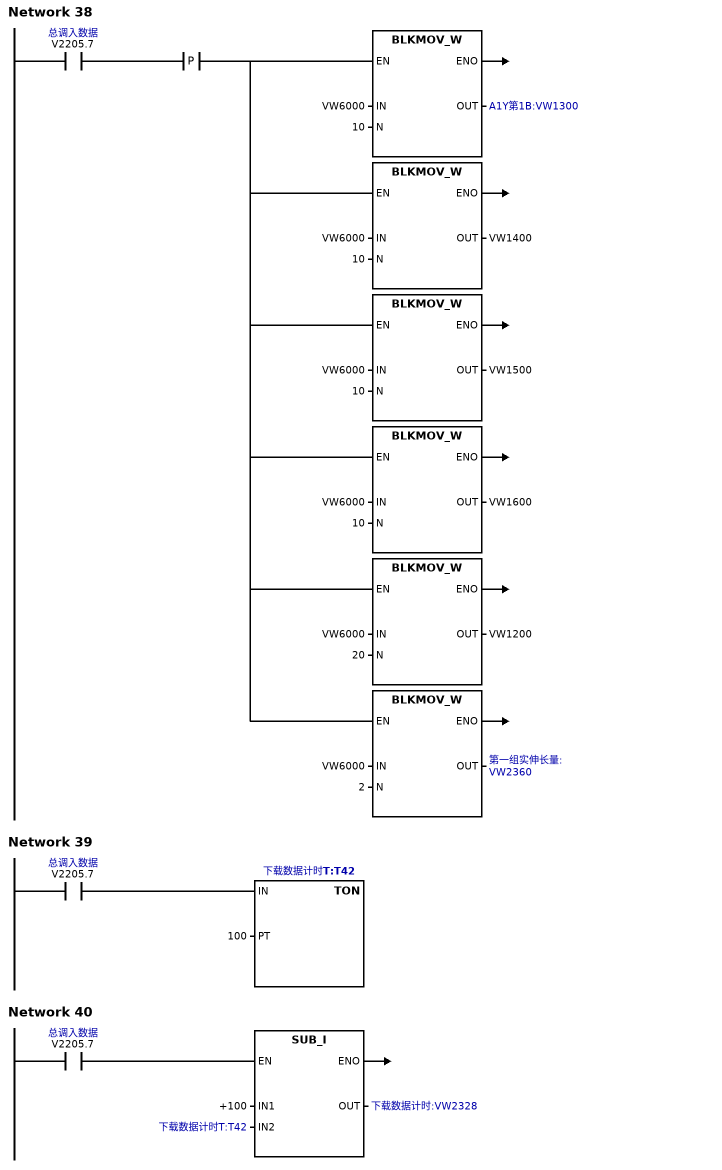
[picture p48: SBR18 networks 38-40]
Network 38
LD     总调入数据:V2205.7
EU
BMW    VW6000, A1Y第1B:VW1300, 10
BMW    VW6000, VW1400, 10
BMW    VW6000, VW1500, 10
BMW    VW6000, VW1600, 10
BMW    VW6000, VW1200, 20
BMW    VW6000, 第一组实伸长量:VW2360, 2
Network 39
LD     总调入数据:V2205.7
TON    下载数据计时T:T42, 100
Network 40
LD     总调入数据:V2205.7
MOVW   +100, 下载数据计时:VW2328
-I     下载数据计时T:T42, 下载数据计时:VW2328
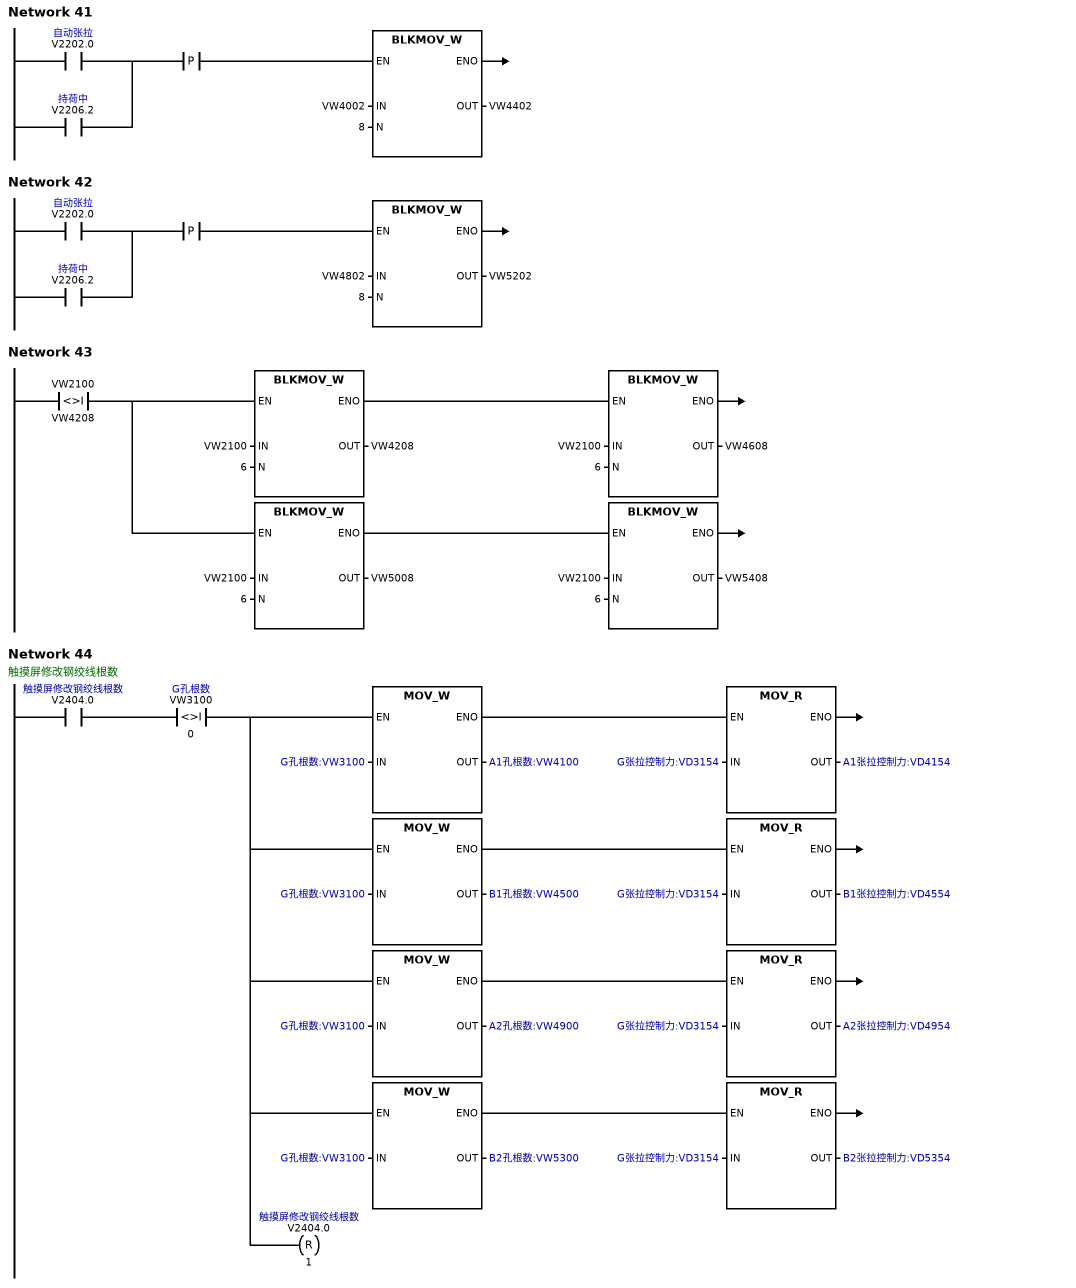
Network 41
LD     自动张拉:V2202.0
O      持荷中:V2206.2
EU
BMW    VW4002, VW4402, 8
Network 42
LD     自动张拉:V2202.0
O      持荷中:V2206.2
EU
BMW    VW4802, VW5202, 8
Network 43
LDW<>  VW2100, VW4208
LPS
BMW    VW2100, VW4208, 6
AENO
BMW    VW2100, VW4608, 6
LPP
BMW    VW2100, VW5008, 6
AENO
BMW    VW2100, VW5408, 6
Network 44
// 触摸屏修改钢绞线根数
LD     触摸屏修改钢绞线根数:V2404.0
AW<>   G孔根数:VW3100, 0
LPS
MOVW   G孔根数:VW3100, A1孔根数:VW4100
AENO
MOVR   G张拉控制力:VD3154, A1张拉控制力:VD4154
LRD
MOVW   G孔根数:VW3100, B1孔根数:VW4500
AENO
MOVR   G张拉控制力:VD3154, B1张拉控制力:VD4554
LRD
MOVW   G孔根数:VW3100, A2孔根数:VW4900
AENO
MOVR   G张拉控制力:VD3154, A2张拉控制力:VD4954
LRD
MOVW   G孔根数:VW3100, B2孔根数:VW5300
AENO
MOVR   G张拉控制力:VD3154, B2张拉控制力:VD5354
LPP
R      触摸屏修改钢绞线根数:V2404.0, 1
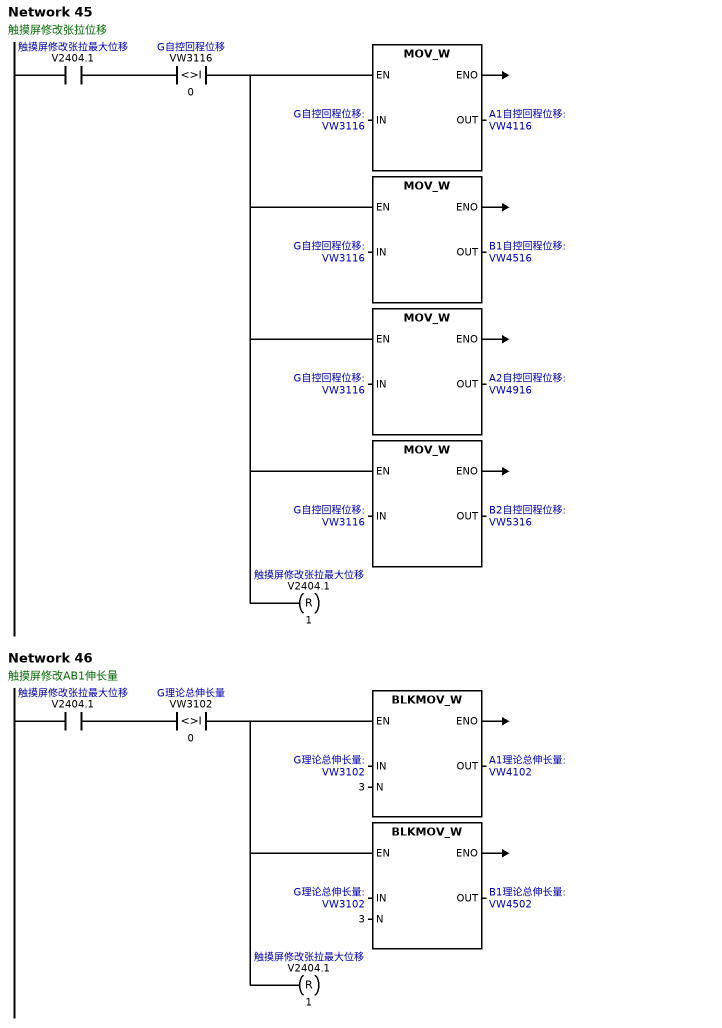
Network 45
// 触摸屏修改张拉位移
LD     触摸屏修改张拉最大位移:V2404.1
AW<>   G自控回程位移:VW3116, 0
MOVW   G自控回程位移:VW3116, A1自控回程位移:VW4116
MOVW   G自控回程位移:VW3116, B1自控回程位移:VW4516
MOVW   G自控回程位移:VW3116, A2自控回程位移:VW4916
MOVW   G自控回程位移:VW3116, B2自控回程位移:VW5316
R      触摸屏修改张拉最大位移:V2404.1, 1
Network 46
// 触摸屏修改AB1伸长量
LD     触摸屏修改张拉最大位移:V2404.1
AW<>   G理论总伸长量:VW3102, 0
BMW    G理论总伸长量:VW3102, A1理论总伸长量:VW4102, 3
BMW    G理论总伸长量:VW3102, B1理论总伸长量:VW4502, 3
R      触摸屏修改张拉最大位移:V2404.1, 1
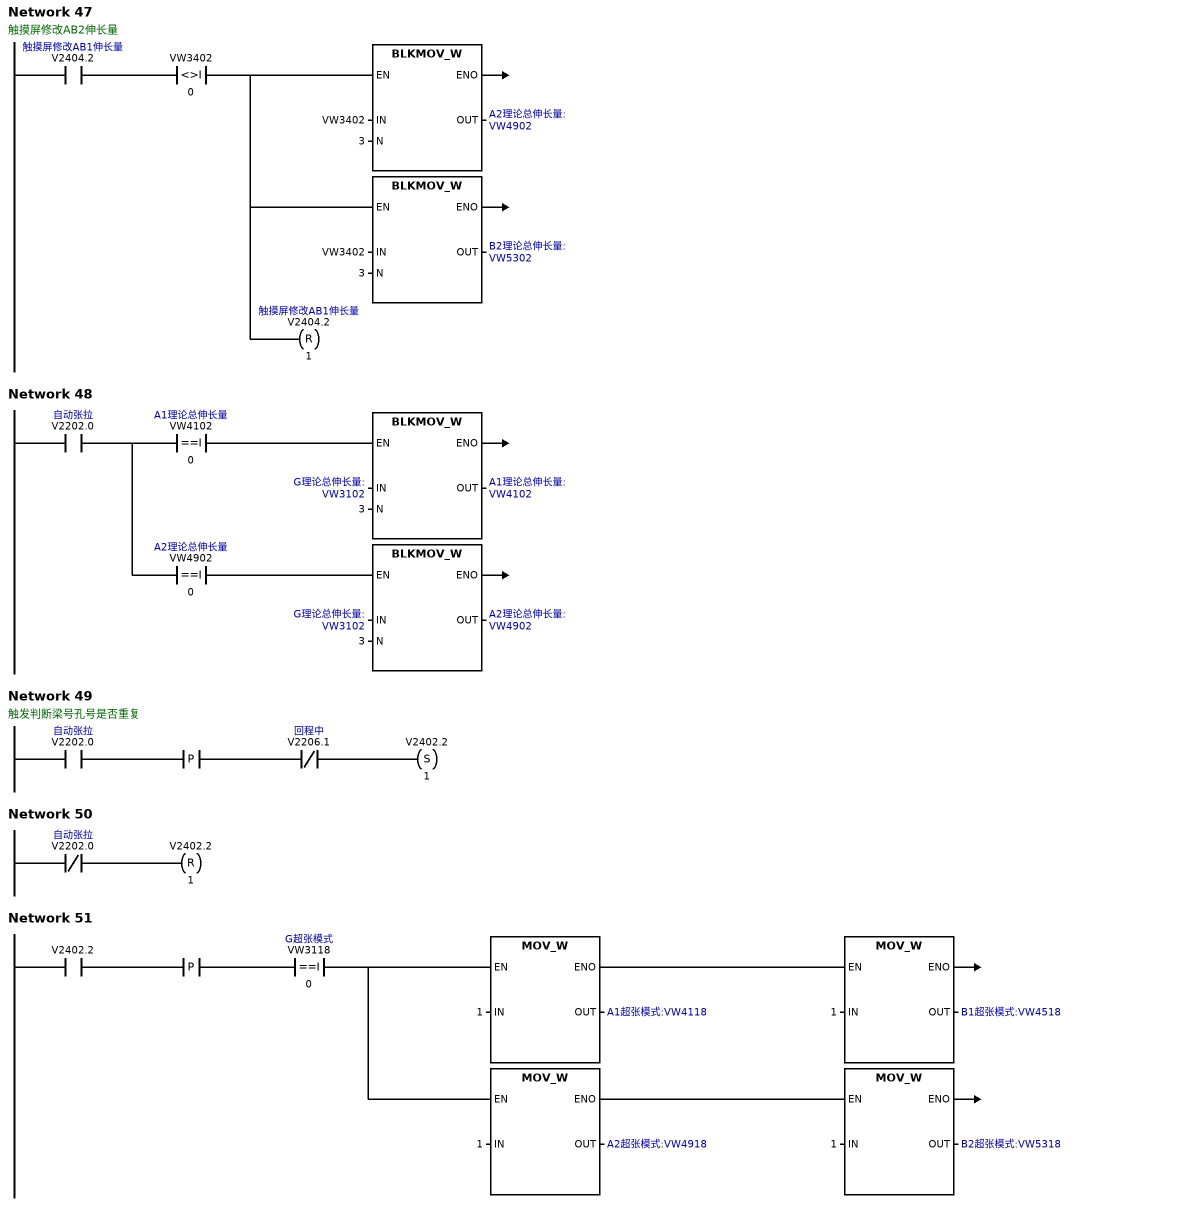
Network 47
// 触摸屏修改AB2伸长量
LD     触摸屏修改AB1伸长量:V2404.2
AW<>   VW3402, 0
BMW    VW3402, A2理论总伸长量:VW4902, 3
BMW    VW3402, B2理论总伸长量:VW5302, 3
R      触摸屏修改AB1伸长量:V2404.2, 1
Network 48
LD     自动张拉:V2202.0
LPS
AW=    A1理论总伸长量:VW4102, 0
BMW    G理论总伸长量:VW3102, A1理论总伸长量:VW4102, 3
LPP
AW=    A2理论总伸长量:VW4902, 0
BMW    G理论总伸长量:VW3102, A2理论总伸长量:VW4902, 3
Network 49
// 触发判断梁号孔号是否重复
LD     自动张拉:V2202.0
EU
AN     回程中:V2206.1
S      V2402.2, 1
Network 50
LDN    自动张拉:V2202.0
R      V2402.2, 1
Network 51
LD     V2402.2
EU
AW=    G超张模式:VW3118, 0
LPS
MOVW   1, A1超张模式:VW4118
AENO
MOVW   1, B1超张模式:VW4518
LPP
MOVW   1, A2超张模式:VW4918
AENO
MOVW   1, B2超张模式:VW5318
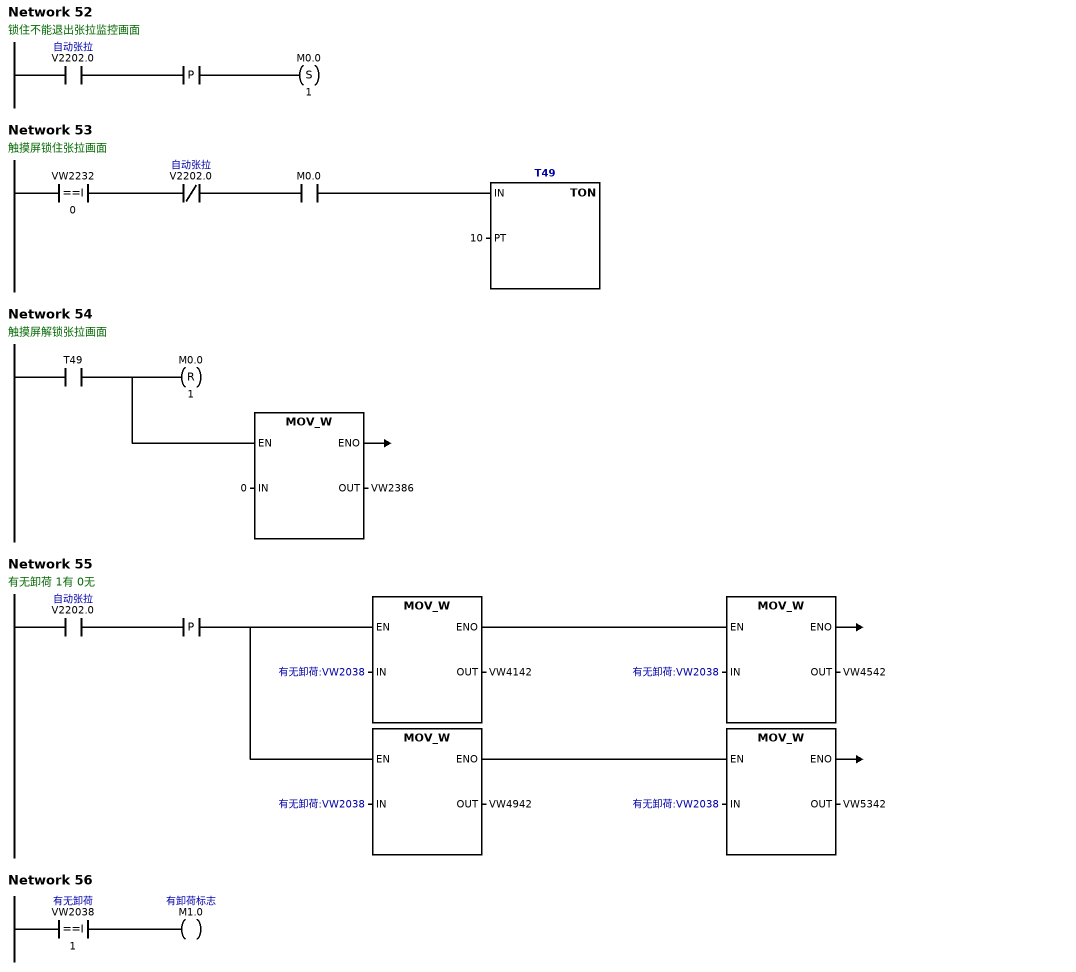
Network 52
// 锁住不能退出张拉监控画面
LD     自动张拉:V2202.0
EU
S      M0.0, 1
Network 53
// 触摸屏锁住张拉画面
LDW=   VW2232, 0
AN     自动张拉:V2202.0
A      M0.0
TON    T49, 10
Network 54
// 触摸屏解锁张拉画面
LD     T49
R      M0.0, 1
MOVW   0, VW2386
Network 55
// 有无卸荷 1有 0无
LD     自动张拉:V2202.0
EU
LPS
MOVW   有无卸荷:VW2038, VW4142
AENO
MOVW   有无卸荷:VW2038, VW4542
LPP
MOVW   有无卸荷:VW2038, VW4942
AENO
MOVW   有无卸荷:VW2038, VW5342
Network 56
LDW=   有无卸荷:VW2038, 1
=      有卸荷标志:M1.0
END_SUBROUTINE_BLOCK

SUBROUTINE_BLOCK A1自动控制:SBR19
TITLE=子程序注释
VAR
目标压力下限:INT;	// LW0 
目标压力上限:INT;	// LW2 
比较位移:INT;	// LW4 
与比较位移的差值:INT;	// LW6 
END_VAR
BEGIN
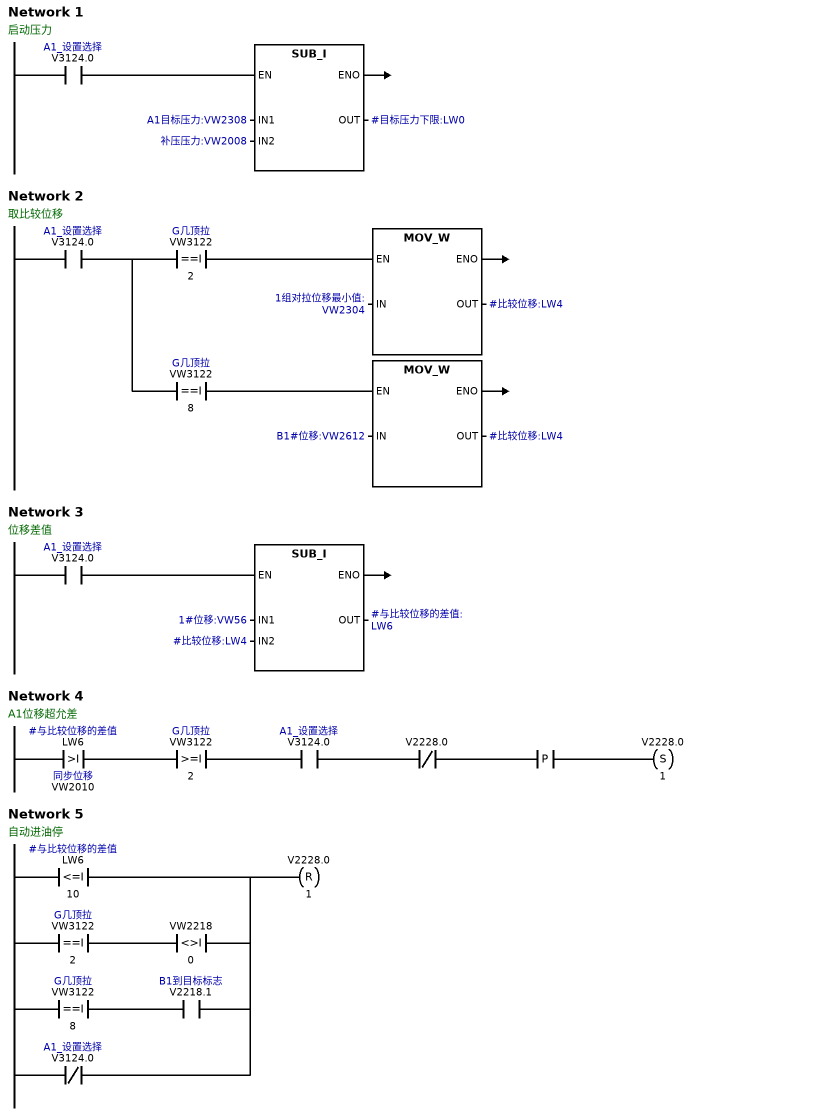
Network 1
// 启动压力
LD     A1_设置选择:V3124.0
MOVW   A1目标压力:VW2308, #目标压力下限:LW0
-I     补压压力:VW2008, #目标压力下限:LW0
Network 2
// 取比较位移
LD     A1_设置选择:V3124.0
LPS
AW=    G几顶拉:VW3122, 2
MOVW   1组对拉位移最小值:VW2304, #比较位移:LW4
LPP
AW=    G几顶拉:VW3122, 8
MOVW   B1#位移:VW2612, #比较位移:LW4
Network 3
// 位移差值
LD     A1_设置选择:V3124.0
MOVW   1#位移:VW56, #与比较位移的差值:LW6
-I     #比较位移:LW4, #与比较位移的差值:LW6
Network 4
// A1位移超允差
LDW>   #与比较位移的差值:LW6, 同步位移:VW2010
AW>=   G几顶拉:VW3122, 2
A      A1_设置选择:V3124.0
AN     V2228.0
EU
S      V2228.0, 1
Network 5
// 自动进油停
LDW<=  #与比较位移的差值:LW6, 10
LDW=   G几顶拉:VW3122, 2
AW<>   VW2218, 0
OLD
LDW=   G几顶拉:VW3122, 8
A      B1到目标标志:V2218.1
OLD
ON     A1_设置选择:V3124.0
R      V2228.0, 1
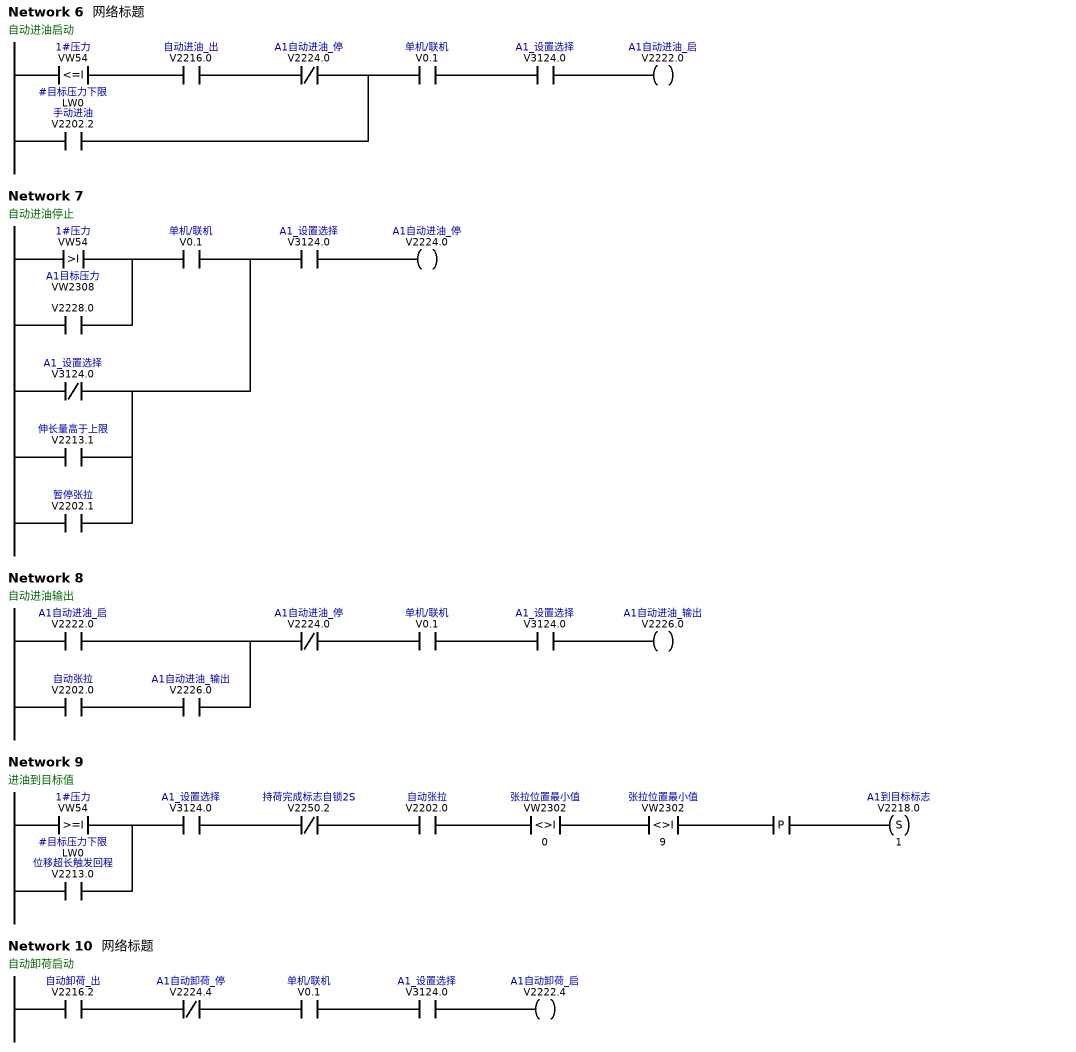
Network 6 // 网络标题
// 自动进油启动
LDW<=  1#压力:VW54, #目标压力下限:LW0
A      自动进油_出:V2216.0
AN     A1自动进油_停:V2224.0
O      手动进油:V2202.2
A      单机/联机:V0.1
A      A1_设置选择:V3124.0
=      A1自动进油_启:V2222.0
Network 7
// 自动进油停止
LDW>   1#压力:VW54, A1目标压力:VW2308
O      V2228.0
A      单机/联机:V0.1
LDN    A1_设置选择:V3124.0
O      伸长量高于上限:V2213.1
O      暂停张拉:V2202.1
OLD
A      A1_设置选择:V3124.0
=      A1自动进油_停:V2224.0
Network 8
// 自动进油输出
LD     A1自动进油_启:V2222.0
LD     自动张拉:V2202.0
A      A1自动进油_输出:V2226.0
OLD
AN     A1自动进油_停:V2224.0
A      单机/联机:V0.1
A      A1_设置选择:V3124.0
=      A1自动进油_输出:V2226.0
Network 9
// 进油到目标值
LDW>=  1#压力:VW54, #目标压力下限:LW0
O      位移超长触发回程:V2213.0
A      A1_设置选择:V3124.0
AN     持荷完成标志自锁2S:V2250.2
A      自动张拉:V2202.0
AW<>   张拉位置最小值:VW2302, 0
AW<>   张拉位置最小值:VW2302, 9
EU
S      A1到目标标志:V2218.0, 1
Network 10 // 网络标题
// 自动卸荷启动
LD     自动卸荷_出:V2216.2
AN     A1自动卸荷_停:V2224.4
A      单机/联机:V0.1
A      A1_设置选择:V3124.0
=      A1自动卸荷_启:V2222.4
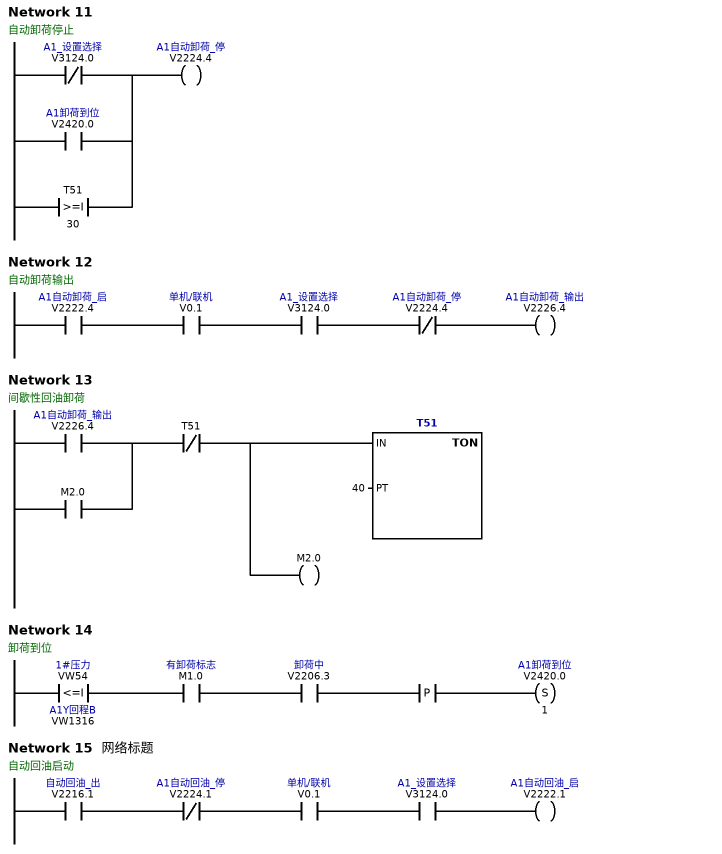
Network 11
// 自动卸荷停止
LDN    A1_设置选择:V3124.0
O      A1卸荷到位:V2420.0
OW>=   T51, 30
=      A1自动卸荷_停:V2224.4
Network 12
// 自动卸荷输出
LD     A1自动卸荷_启:V2222.4
A      单机/联机:V0.1
A      A1_设置选择:V3124.0
AN     A1自动卸荷_停:V2224.4
=      A1自动卸荷_输出:V2226.4
Network 13
// 间歇性回油卸荷
LD     A1自动卸荷_输出:V2226.4
O      M2.0
AN     T51
TON    T51, 40
=      M2.0
Network 14
// 卸荷到位
LDW<=  1#压力:VW54, A1Y回程B:VW1316
A      有卸荷标志:M1.0
A      卸荷中:V2206.3
EU
S      A1卸荷到位:V2420.0, 1
Network 15 // 网络标题
// 自动回油启动
LD     自动回油_出:V2216.1
AN     A1自动回油_停:V2224.1
A      单机/联机:V0.1
A      A1_设置选择:V3124.0
=      A1自动回油_启:V2222.1
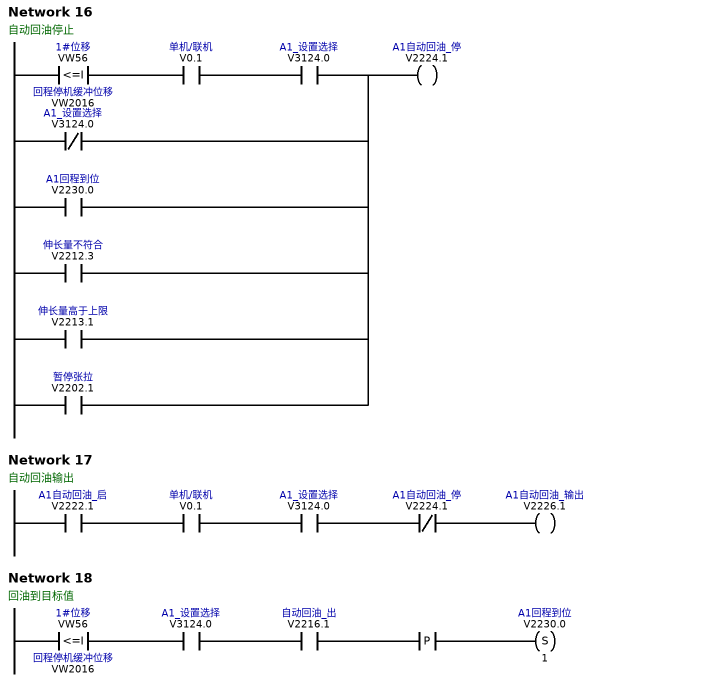
Network 16
// 自动回油停止
LDW<=  1#位移:VW56, 回程停机缓冲位移:VW2016
A      单机/联机:V0.1
A      A1_设置选择:V3124.0
ON     A1_设置选择:V3124.0
O      A1回程到位:V2230.0
O      伸长量不符合:V2212.3
O      伸长量高于上限:V2213.1
O      暂停张拉:V2202.1
=      A1自动回油_停:V2224.1
Network 17
// 自动回油输出
LD     A1自动回油_启:V2222.1
A      单机/联机:V0.1
A      A1_设置选择:V3124.0
AN     A1自动回油_停:V2224.1
=      A1自动回油_输出:V2226.1
Network 18
// 回油到目标值
LDW<=  1#位移:VW56, 回程停机缓冲位移:VW2016
A      A1_设置选择:V3124.0
A      自动回油_出:V2216.1
EU
S      A1回程到位:V2230.0, 1
END_SUBROUTINE_BLOCK

SUBROUTINE_BLOCK A2自动控制:SBR20
TITLE=
VAR
目标压力下限:INT;	// LW0 
目标压力上限:INT;	// LW2 
比较位移:INT;	// LW4 
与比较位移的差值:INT;	// LW6 
END_VAR
BEGIN
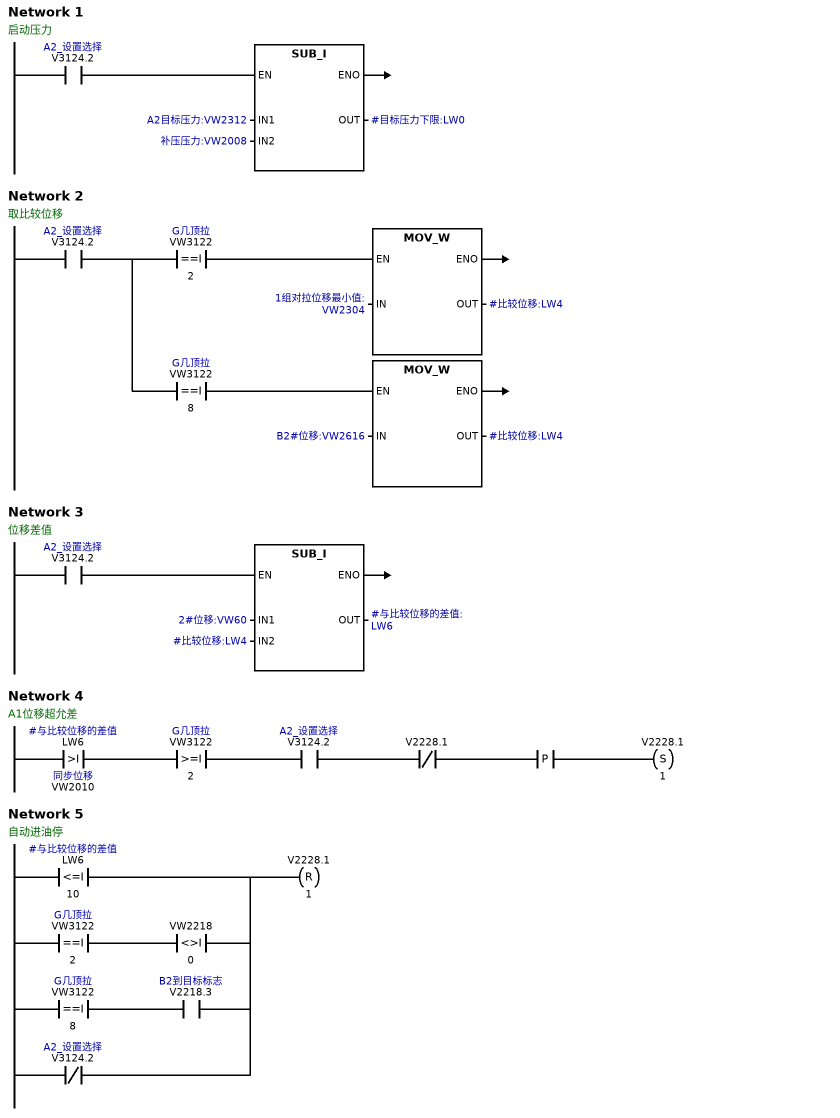
Network 1
// 启动压力
LD     A2_设置选择:V3124.2
MOVW   A2目标压力:VW2312, #目标压力下限:LW0
-I     补压压力:VW2008, #目标压力下限:LW0
Network 2
// 取比较位移
LD     A2_设置选择:V3124.2
LPS
AW=    G几顶拉:VW3122, 2
MOVW   1组对拉位移最小值:VW2304, #比较位移:LW4
LPP
AW=    G几顶拉:VW3122, 8
MOVW   B2#位移:VW2616, #比较位移:LW4
Network 3
// 位移差值
LD     A2_设置选择:V3124.2
MOVW   2#位移:VW60, #与比较位移的差值:LW6
-I     #比较位移:LW4, #与比较位移的差值:LW6
Network 4
// A1位移超允差
LDW>   #与比较位移的差值:LW6, 同步位移:VW2010
AW>=   G几顶拉:VW3122, 2
A      A2_设置选择:V3124.2
AN     V2228.1
EU
S      V2228.1, 1
Network 5
// 自动进油停
LDW<=  #与比较位移的差值:LW6, 10
LDW=   G几顶拉:VW3122, 2
AW<>   VW2218, 0
OLD
LDW=   G几顶拉:VW3122, 8
A      B2到目标标志:V2218.3
OLD
ON     A2_设置选择:V3124.2
R      V2228.1, 1
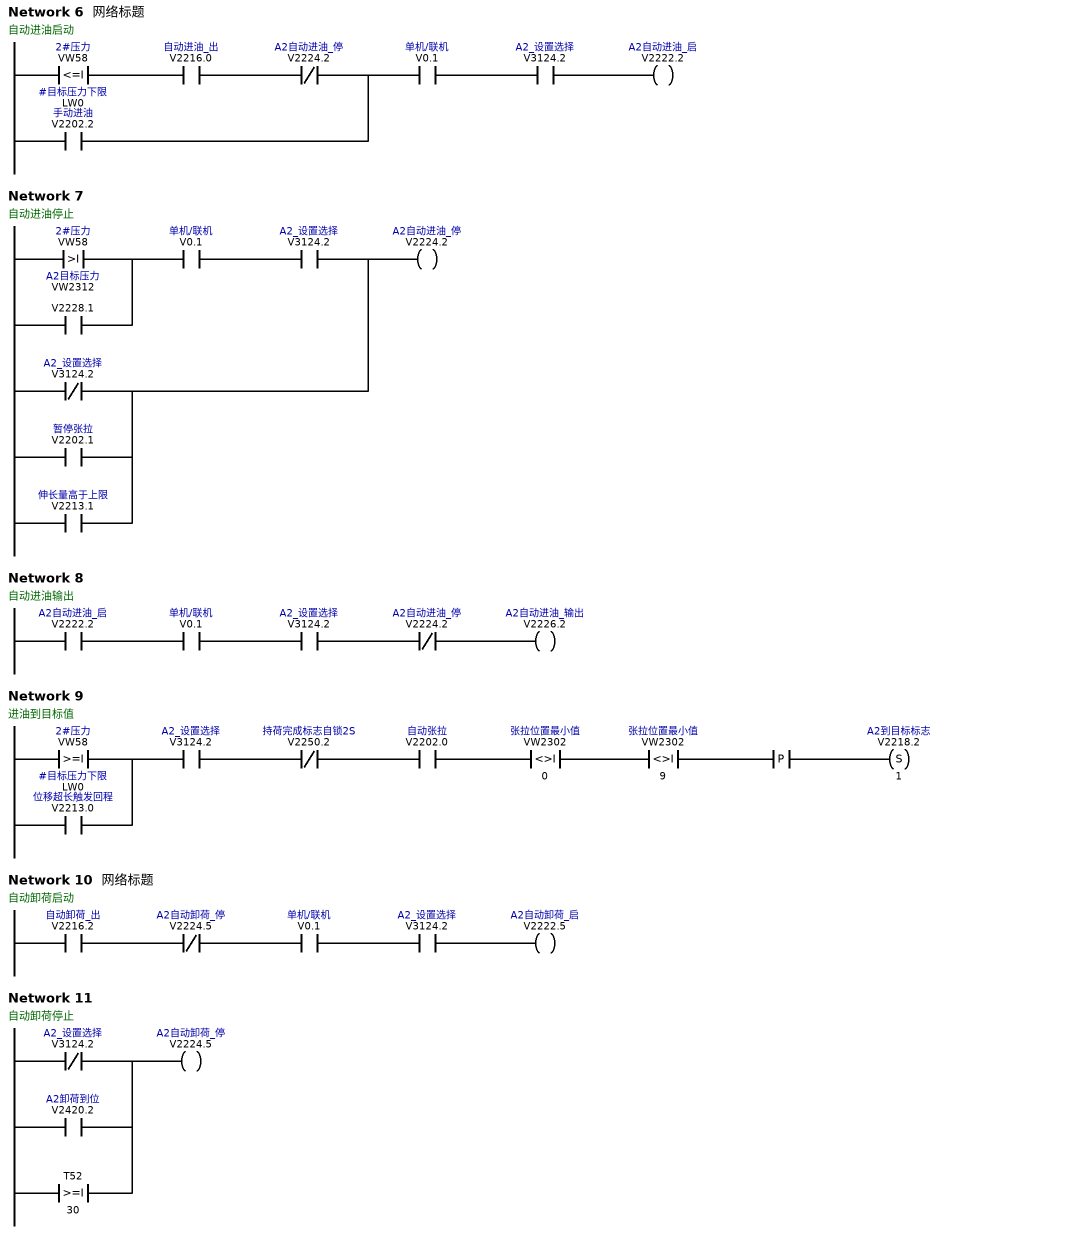
Network 6 // 网络标题
// 自动进油启动
LDW<=  2#压力:VW58, #目标压力下限:LW0
A      自动进油_出:V2216.0
AN     A2自动进油_停:V2224.2
O      手动进油:V2202.2
A      单机/联机:V0.1
A      A2_设置选择:V3124.2
=      A2自动进油_启:V2222.2
Network 7
// 自动进油停止
LDW>   2#压力:VW58, A2目标压力:VW2312
O      V2228.1
A      单机/联机:V0.1
A      A2_设置选择:V3124.2
LDN    A2_设置选择:V3124.2
O      暂停张拉:V2202.1
O      伸长量高于上限:V2213.1
OLD
=      A2自动进油_停:V2224.2
Network 8
// 自动进油输出
LD     A2自动进油_启:V2222.2
A      单机/联机:V0.1
A      A2_设置选择:V3124.2
AN     A2自动进油_停:V2224.2
=      A2自动进油_输出:V2226.2
Network 9
// 进油到目标值
LDW>=  2#压力:VW58, #目标压力下限:LW0
O      位移超长触发回程:V2213.0
A      A2_设置选择:V3124.2
AN     持荷完成标志自锁2S:V2250.2
A      自动张拉:V2202.0
AW<>   张拉位置最小值:VW2302, 0
AW<>   张拉位置最小值:VW2302, 9
EU
S      A2到目标标志:V2218.2, 1
Network 10 // 网络标题
// 自动卸荷启动
LD     自动卸荷_出:V2216.2
AN     A2自动卸荷_停:V2224.5
A      单机/联机:V0.1
A      A2_设置选择:V3124.2
=      A2自动卸荷_启:V2222.5
Network 11
// 自动卸荷停止
LDN    A2_设置选择:V3124.2
O      A2卸荷到位:V2420.2
OW>=   T52, 30
=      A2自动卸荷_停:V2224.5
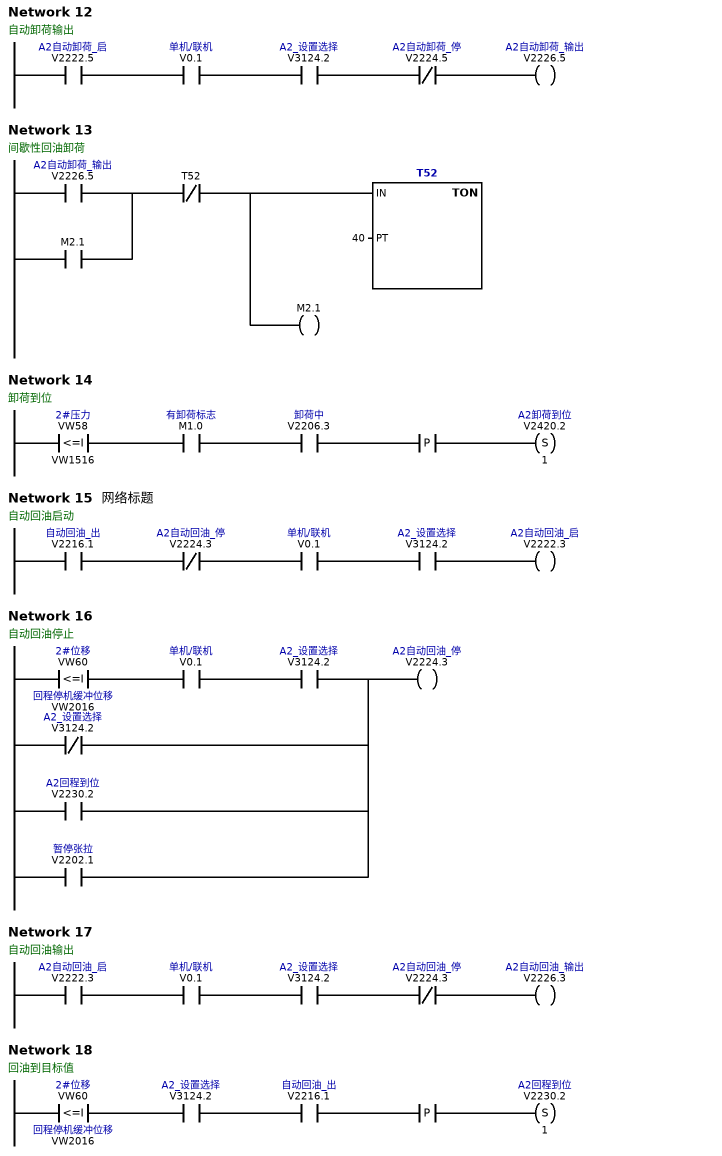
Network 12
// 自动卸荷输出
LD     A2自动卸荷_启:V2222.5
A      单机/联机:V0.1
A      A2_设置选择:V3124.2
AN     A2自动卸荷_停:V2224.5
=      A2自动卸荷_输出:V2226.5
Network 13
// 间歇性回油卸荷
LD     A2自动卸荷_输出:V2226.5
O      M2.1
AN     T52
TON    T52, 40
=      M2.1
Network 14
// 卸荷到位
LDW<=  2#压力:VW58, VW1516
A      有卸荷标志:M1.0
A      卸荷中:V2206.3
EU
S      A2卸荷到位:V2420.2, 1
Network 15 // 网络标题
// 自动回油启动
LD     自动回油_出:V2216.1
AN     A2自动回油_停:V2224.3
A      单机/联机:V0.1
A      A2_设置选择:V3124.2
=      A2自动回油_启:V2222.3
Network 16
// 自动回油停止
LDW<=  2#位移:VW60, 回程停机缓冲位移:VW2016
A      单机/联机:V0.1
A      A2_设置选择:V3124.2
ON     A2_设置选择:V3124.2
O      A2回程到位:V2230.2
O      暂停张拉:V2202.1
=      A2自动回油_停:V2224.3
Network 17
// 自动回油输出
LD     A2自动回油_启:V2222.3
A      单机/联机:V0.1
A      A2_设置选择:V3124.2
AN     A2自动回油_停:V2224.3
=      A2自动回油_输出:V2226.3
Network 18
// 回油到目标值
LDW<=  2#位移:VW60, 回程停机缓冲位移:VW2016
A      A2_设置选择:V3124.2
A      自动回油_出:V2216.1
EU
S      A2回程到位:V2230.2, 1
END_SUBROUTINE_BLOCK

SUBROUTINE_BLOCK 时钟:SBR21
TITLE=
VAR
临时变量:INT;	// LW0 
END_VAR
BEGIN
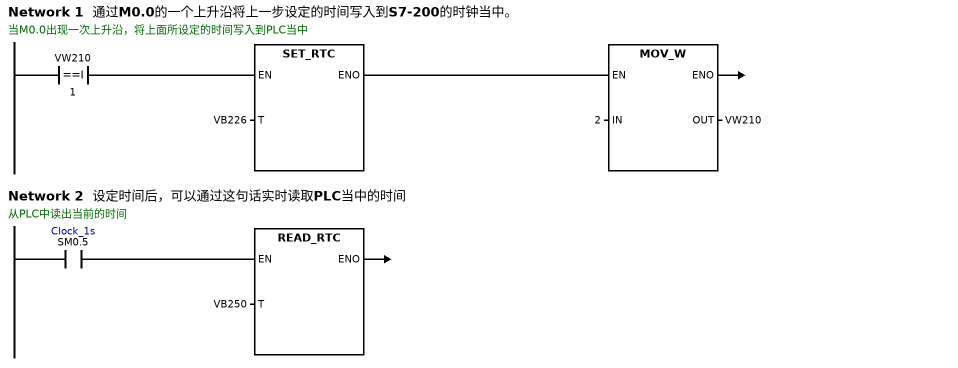
Network 1 // 通过M0.0的一个上升沿将上一步设定的时间写入到S7-200的时钟当中。
// 当M0.0出现一次上升沿，将上面所设定的时间写入到PLC当中
LDW=   VW210, 1
TODW   VB226
AENO
MOVW   2, VW210
Network 2 // 设定时间后，可以通过这句话实时读取PLC当中的时间
// 从PLC中读出当前的时间
LD     Clock_1s:SM0.5
TODR   VB250
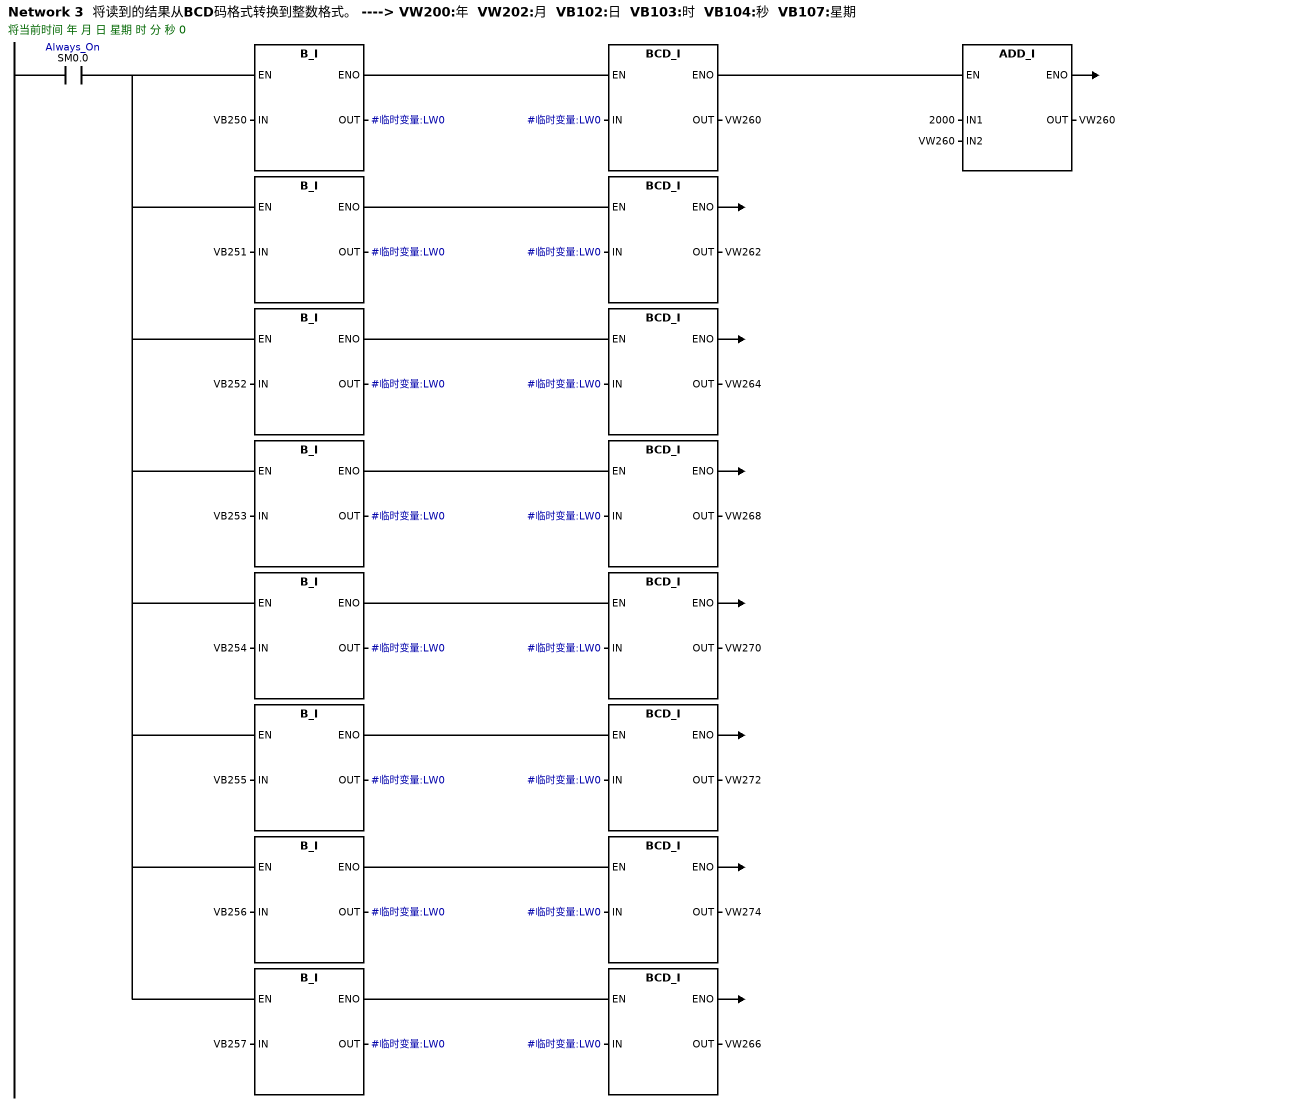
Network 3 // 将读到的结果从BCD码格式转换到整数格式。
----> VW200:年  VW202:月  VB102:日  VB103:时  VB104:秒  VB107:星期  
// 将当前时间 年 月 日 星期 时 分 秒 0
LD     Always_On:SM0.0
LPS
BTI    VB250, #临时变量:LW0
AENO
MOVW   #临时变量:LW0, VW260
AENO
BCDI   VW260
AENO
+I     2000, VW260
LRD
BTI    VB251, #临时变量:LW0
AENO
MOVW   #临时变量:LW0, VW262
BCDI   VW262
LRD
BTI    VB252, #临时变量:LW0
AENO
MOVW   #临时变量:LW0, VW264
BCDI   VW264
LRD
BTI    VB253, #临时变量:LW0
AENO
MOVW   #临时变量:LW0, VW268
BCDI   VW268
LRD
BTI    VB254, #临时变量:LW0
AENO
MOVW   #临时变量:LW0, VW270
BCDI   VW270
LRD
BTI    VB255, #临时变量:LW0
AENO
MOVW   #临时变量:LW0, VW272
BCDI   VW272
LRD
BTI    VB256, #临时变量:LW0
AENO
MOVW   #临时变量:LW0, VW274
BCDI   VW274
LPP
BTI    VB257, #临时变量:LW0
AENO
MOVW   #临时变量:LW0, VW266
BCDI   VW266
END_SUBROUTINE_BLOCK

SUBROUTINE_BLOCK mm:SBR22
TITLE=
VAR
A1:WORD;	// LW0 
A2:WORD;	// LW2 
A3:WORD;	// LW4 
B1:WORD;	// LW6 
B2:WORD;	// LW8 
B3:WORD;	// LW10 
MM1:WORD;	// LW12 
XY1:WORD;	// LW14 
XY2:DINT;	// LD16 
年计算:WORD;	// LW20 
月计算:WORD;	// LW22 
日计算:WORD;	// LW24 
日存:WORD;	// LW26 
月存:WORD;	// LW28 
有效年期:WORD;	// LW30 
END_VAR
BEGIN
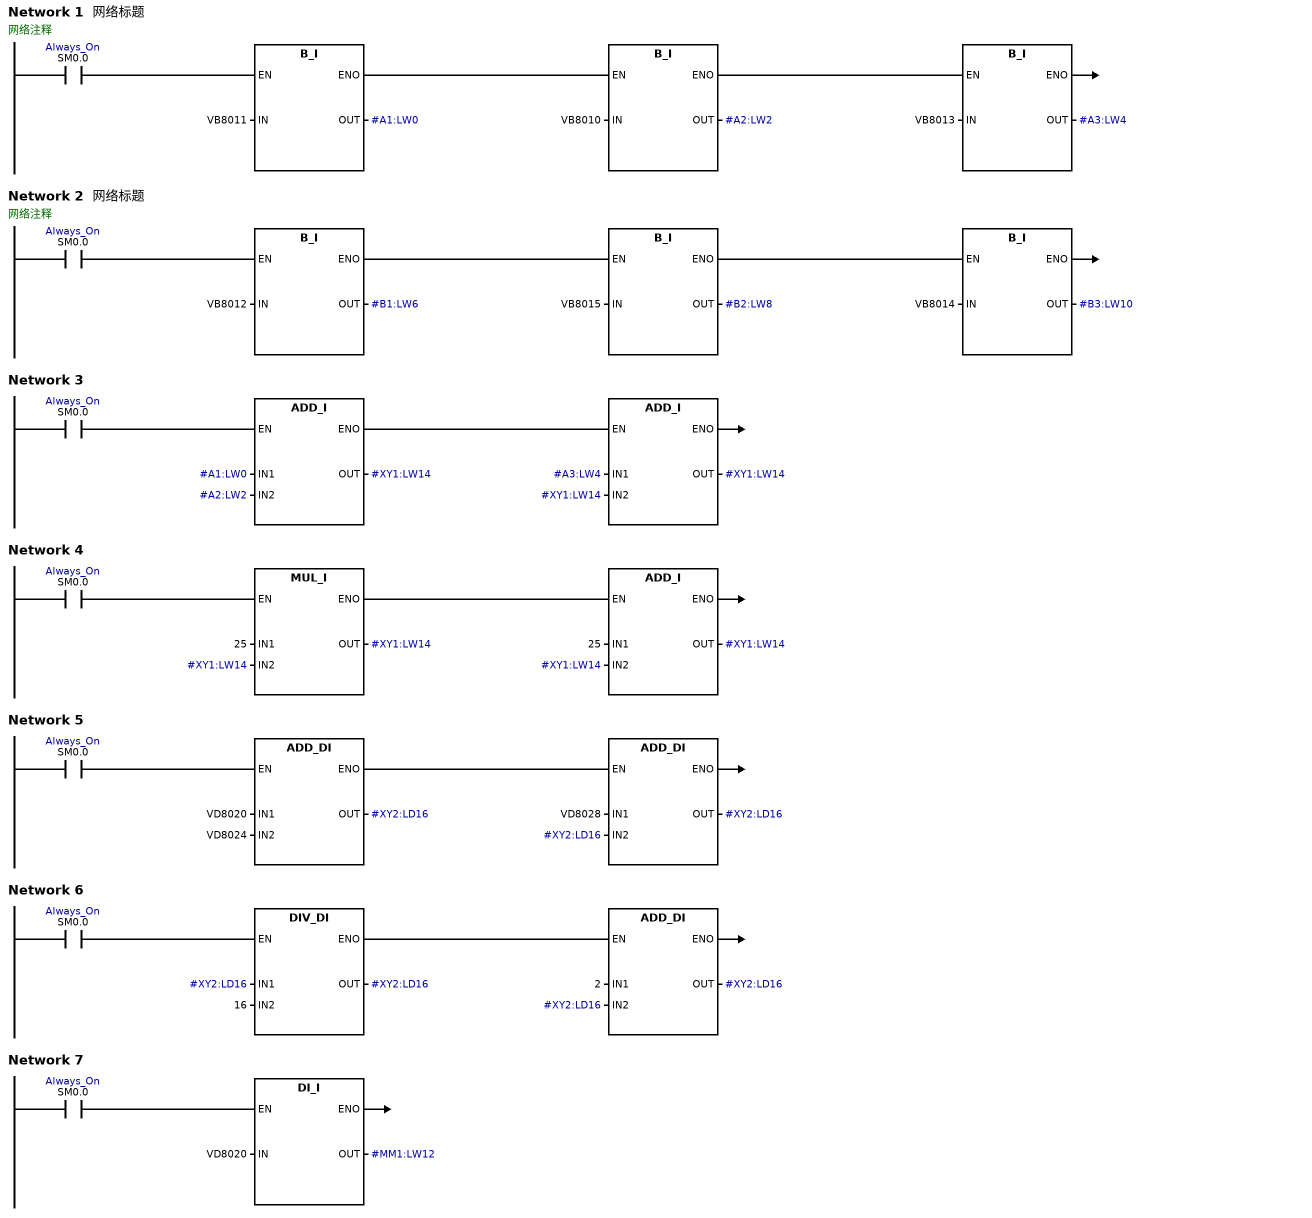
Network 1 // 网络标题
// 网络注释
LD     Always_On:SM0.0
BTI    VB8011, #A1:LW0
AENO
BTI    VB8010, #A2:LW2
AENO
BTI    VB8013, #A3:LW4
Network 2 // 网络标题
// 网络注释
LD     Always_On:SM0.0
BTI    VB8012, #B1:LW6
AENO
BTI    VB8015, #B2:LW8
AENO
BTI    VB8014, #B3:LW10
Network 3
LD     Always_On:SM0.0
MOVW   #A1:LW0, #XY1:LW14
AENO
+I     #A2:LW2, #XY1:LW14
AENO
+I     #A3:LW4, #XY1:LW14
Network 4
LD     Always_On:SM0.0
*I     25, #XY1:LW14
AENO
+I     25, #XY1:LW14
Network 5
LD     Always_On:SM0.0
MOVD   VD8020, #XY2:LD16
AENO
+D     VD8024, #XY2:LD16
AENO
+D     VD8028, #XY2:LD16
Network 6
LD     Always_On:SM0.0
/D     16, #XY2:LD16
AENO
+D     2, #XY2:LD16
Network 7
LD     Always_On:SM0.0
DTI    VD8020, #MM1:LW12
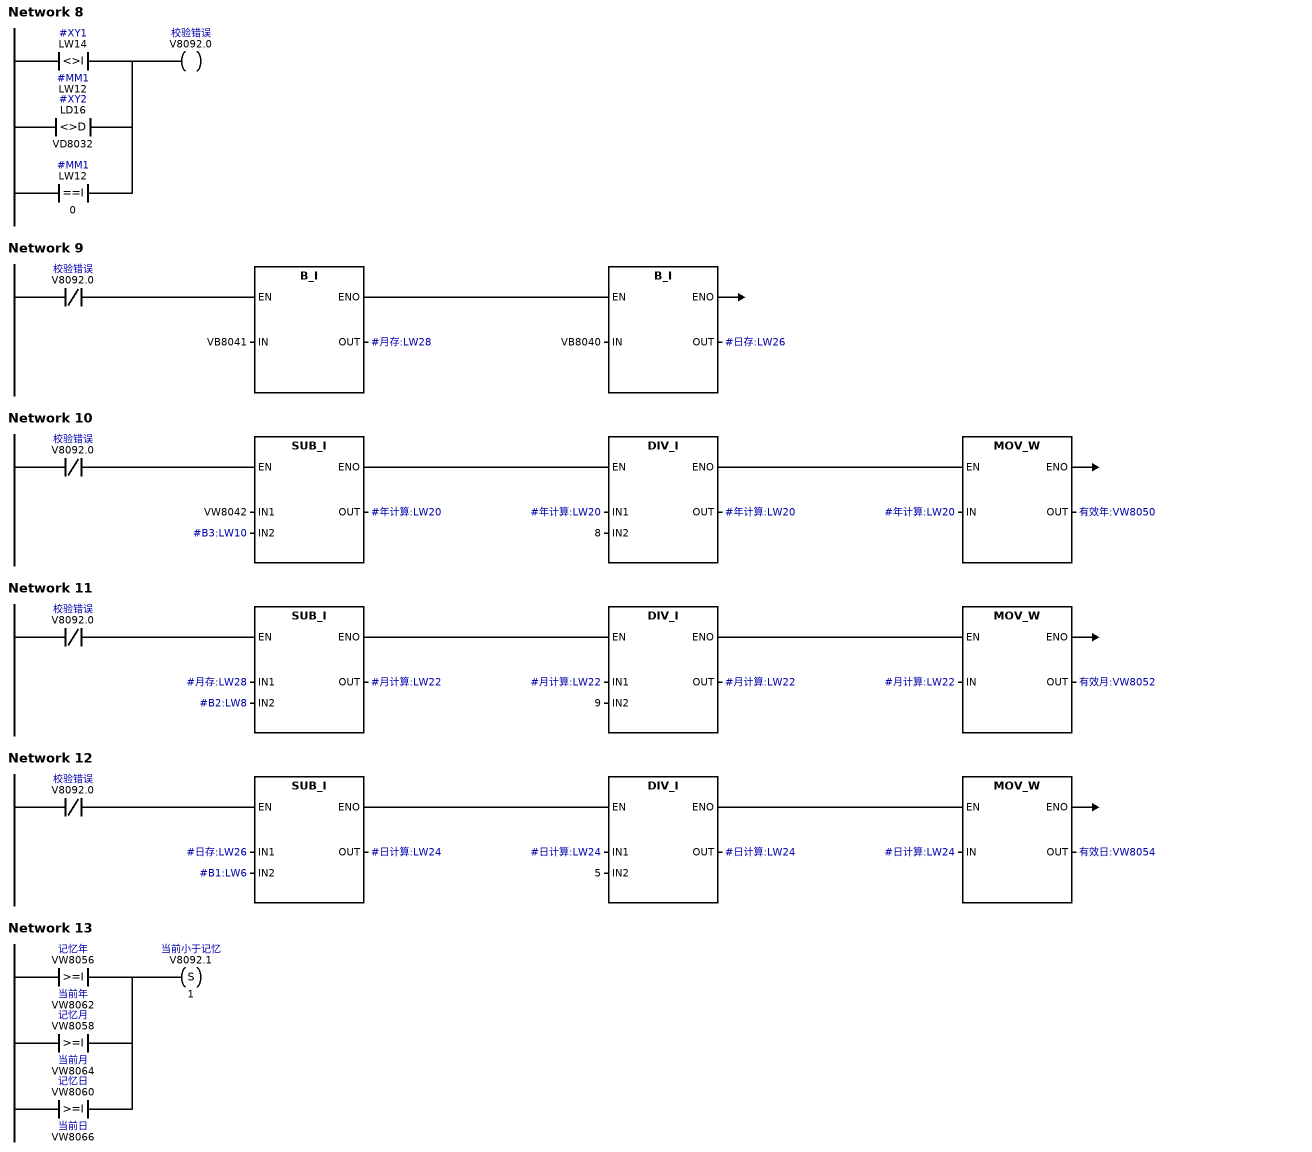
Network 8
LDW<>  #XY1:LW14, #MM1:LW12
OD<>   #XY2:LD16, VD8032
OW=    #MM1:LW12, 0
=      校验错误:V8092.0
Network 9
LDN    校验错误:V8092.0
BTI    VB8041, #月存:LW28
AENO
BTI    VB8040, #日存:LW26
Network 10
LDN    校验错误:V8092.0
MOVW   VW8042, #年计算:LW20
AENO
-I     #B3:LW10, #年计算:LW20
AENO
/I     8, #年计算:LW20
AENO
MOVW   #年计算:LW20, 有效年:VW8050
Network 11
LDN    校验错误:V8092.0
MOVW   #月存:LW28, #月计算:LW22
AENO
-I     #B2:LW8, #月计算:LW22
AENO
/I     9, #月计算:LW22
AENO
MOVW   #月计算:LW22, 有效月:VW8052
Network 12
LDN    校验错误:V8092.0
MOVW   #日存:LW26, #日计算:LW24
AENO
-I     #B1:LW6, #日计算:LW24
AENO
/I     5, #日计算:LW24
AENO
MOVW   #日计算:LW24, 有效日:VW8054
Network 13
LDW>=  记忆年:VW8056, 当前年:VW8062
OW>=   记忆月:VW8058, 当前月:VW8064
OW>=   记忆日:VW8060, 当前日:VW8066
S      当前小于记忆:V8092.1, 1
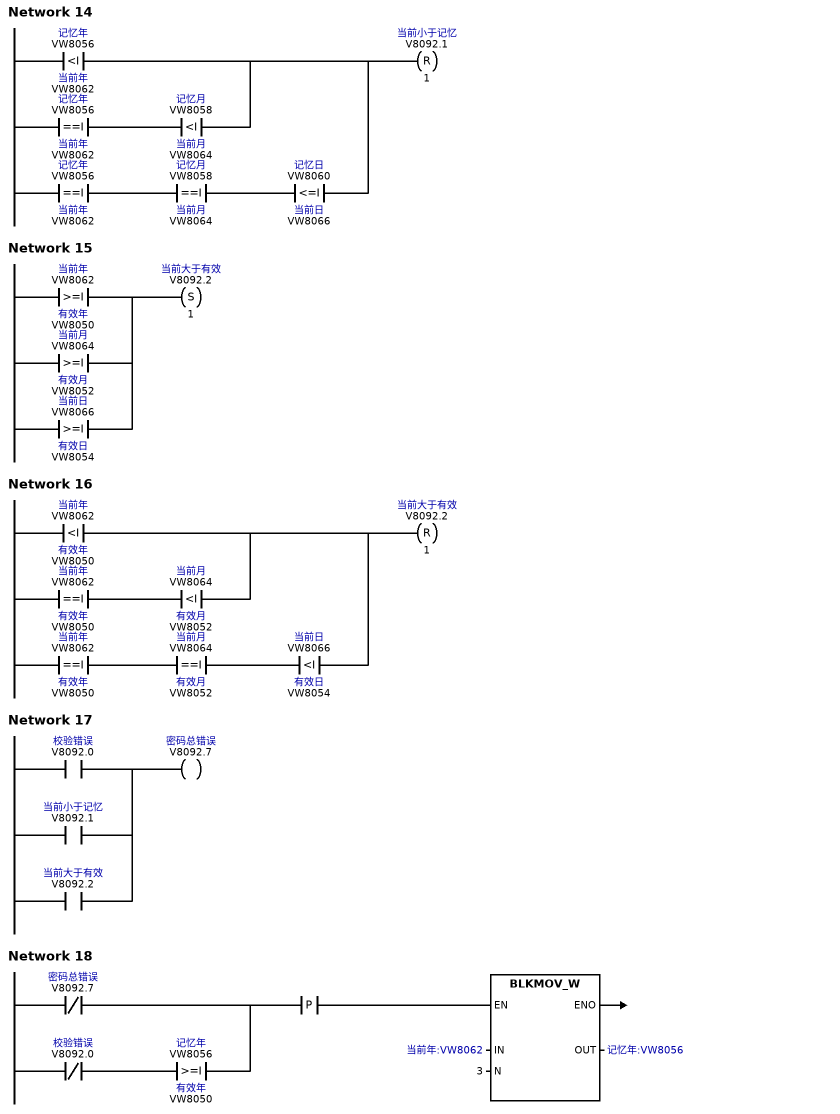
Network 14
LDW<   记忆年:VW8056, 当前年:VW8062
LDW=   记忆年:VW8056, 当前年:VW8062
AW<    记忆月:VW8058, 当前月:VW8064
OLD
LDW=   记忆年:VW8056, 当前年:VW8062
AW=    记忆月:VW8058, 当前月:VW8064
AW<=   记忆日:VW8060, 当前日:VW8066
OLD
R      当前小于记忆:V8092.1, 1
Network 15
LDW>=  当前年:VW8062, 有效年:VW8050
OW>=   当前月:VW8064, 有效月:VW8052
OW>=   当前日:VW8066, 有效日:VW8054
S      当前大于有效:V8092.2, 1
Network 16
LDW<   当前年:VW8062, 有效年:VW8050
LDW=   当前年:VW8062, 有效年:VW8050
AW<    当前月:VW8064, 有效月:VW8052
OLD
LDW=   当前年:VW8062, 有效年:VW8050
AW=    当前月:VW8064, 有效月:VW8052
AW<    当前日:VW8066, 有效日:VW8054
OLD
R      当前大于有效:V8092.2, 1
Network 17
LD     校验错误:V8092.0
O      当前小于记忆:V8092.1
O      当前大于有效:V8092.2
=      密码总错误:V8092.7
Network 18
LDN    密码总错误:V8092.7
LDN    校验错误:V8092.0
AW>=   记忆年:VW8056, 有效年:VW8050
OLD
EU
BMW    当前年:VW8062, 记忆年:VW8056, 3
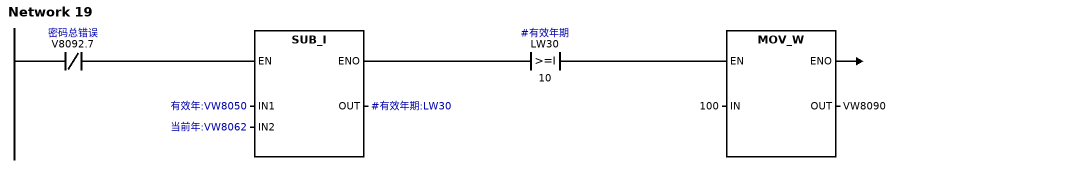
Network 19
LDN    密码总错误:V8092.7
MOVW   有效年:VW8050, #有效年期:LW30
AENO
-I     当前年:VW8062, #有效年期:LW30
AENO
AW>=   #有效年期:LW30, 10
MOVW   100, VW8090
END_SUBROUTINE_BLOCK

SUBROUTINE_BLOCK 主副交换:SBR23
TITLE=子程序注释
BEGIN
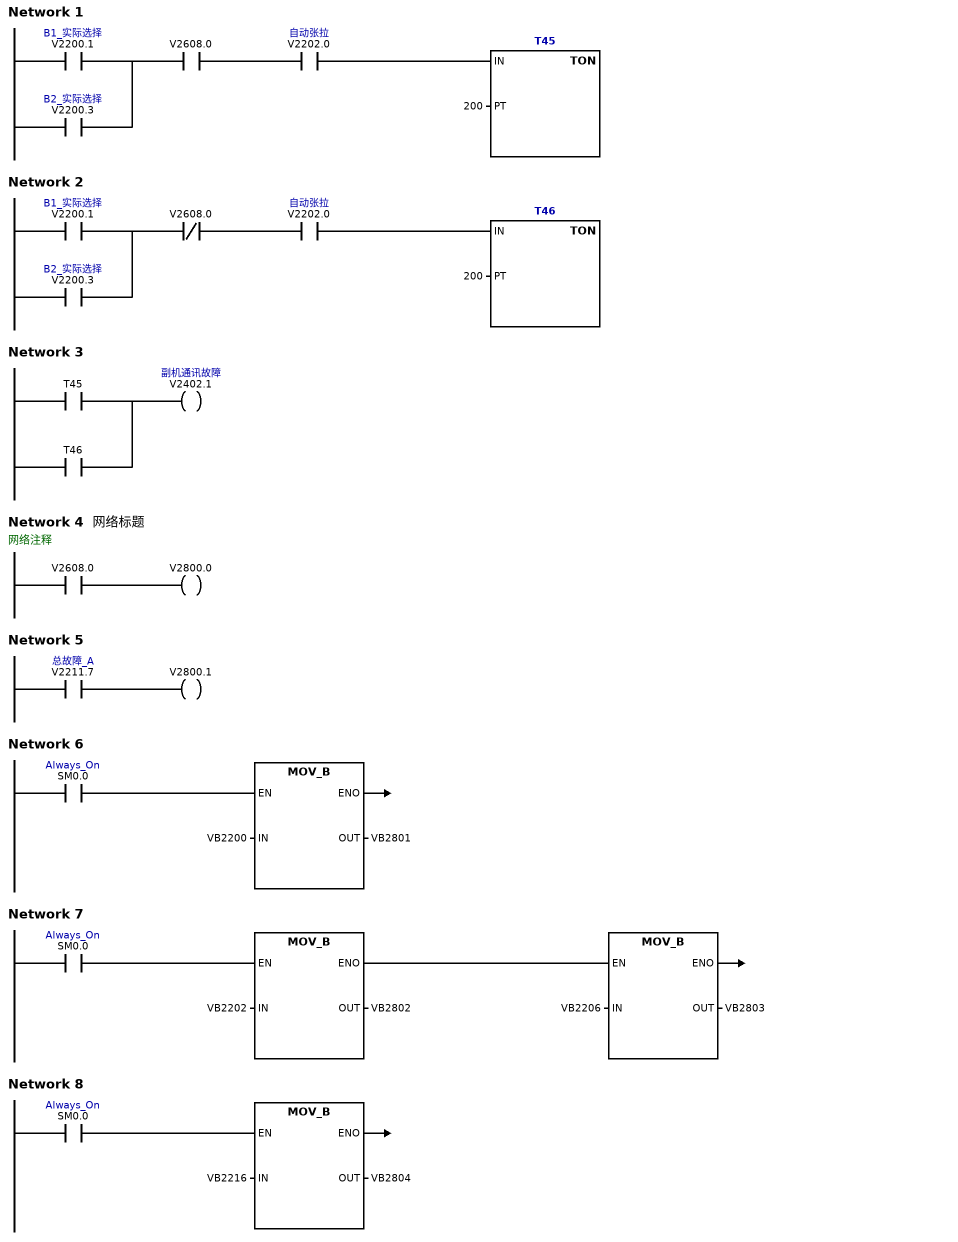
Network 1
LD     B1_实际选择:V2200.1
O      B2_实际选择:V2200.3
A      V2608.0
A      自动张拉:V2202.0
TON    T45, 200
Network 2
LD     B1_实际选择:V2200.1
O      B2_实际选择:V2200.3
AN     V2608.0
A      自动张拉:V2202.0
TON    T46, 200
Network 3
LD     T45
O      T46
=      副机通讯故障:V2402.1
Network 4 // 网络标题
// 网络注释
LD     V2608.0
=      V2800.0
Network 5
LD     总故障_A:V2211.7
=      V2800.1
Network 6
LD     Always_On:SM0.0
MOVB   VB2200, VB2801
Network 7
LD     Always_On:SM0.0
MOVB   VB2202, VB2802
AENO
MOVB   VB2206, VB2803
Network 8
LD     Always_On:SM0.0
MOVB   VB2216, VB2804
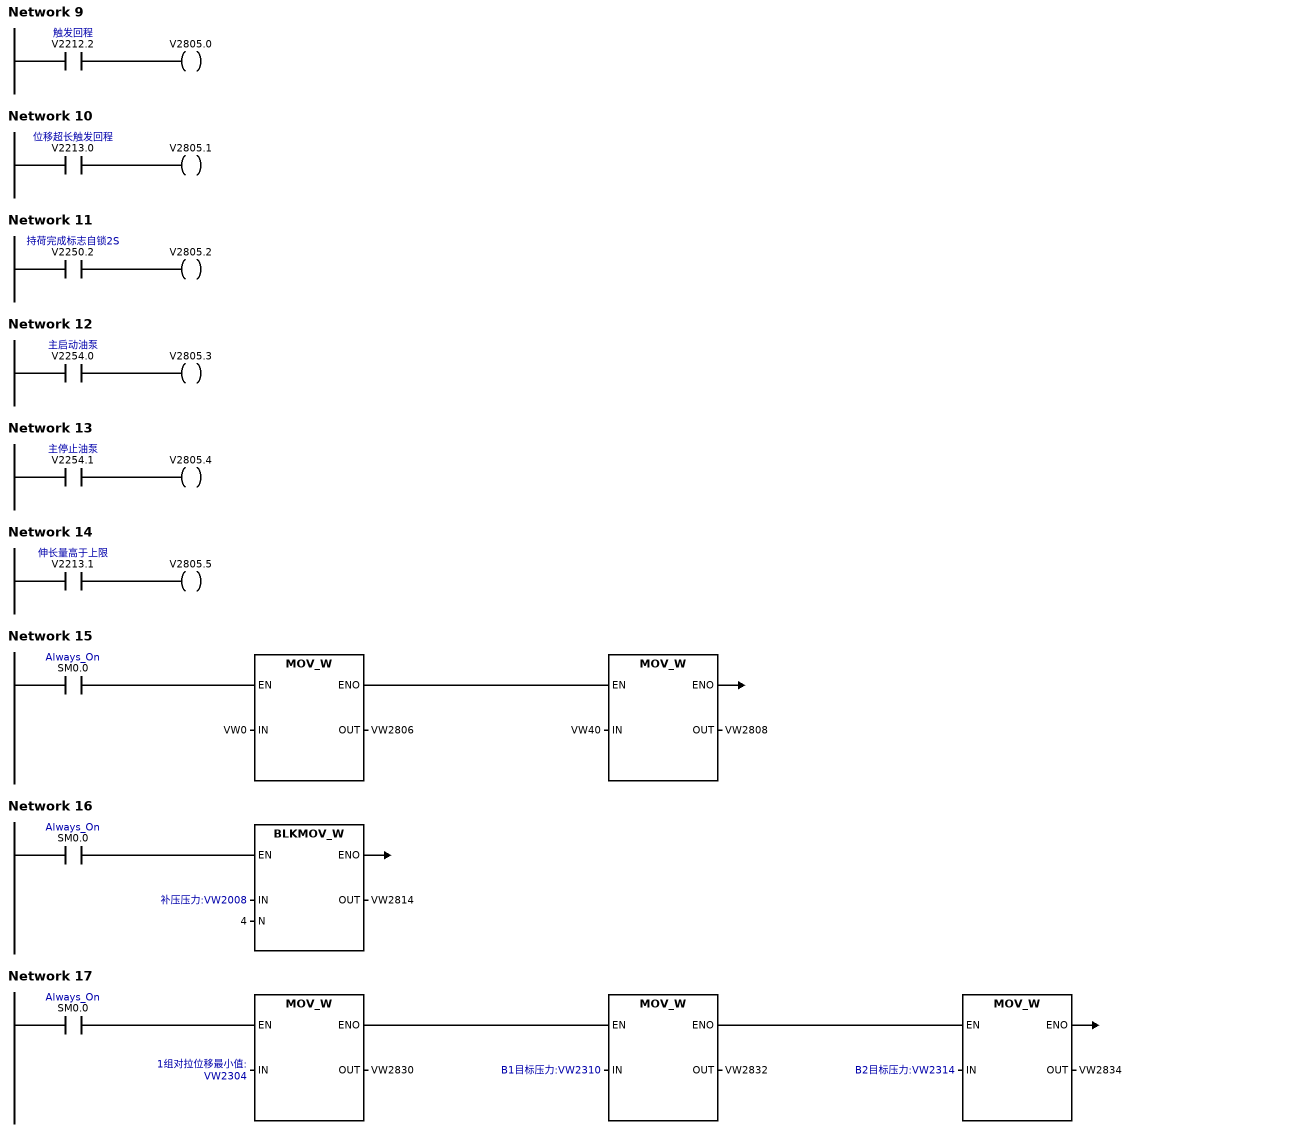
Network 9
LD     触发回程:V2212.2
=      V2805.0
Network 10
LD     位移超长触发回程:V2213.0
=      V2805.1
Network 11
LD     持荷完成标志自锁2S:V2250.2
=      V2805.2
Network 12
LD     主启动油泵:V2254.0
=      V2805.3
Network 13
LD     主停止油泵:V2254.1
=      V2805.4
Network 14
LD     伸长量高于上限:V2213.1
=      V2805.5
Network 15
LD     Always_On:SM0.0
MOVW   VW0, VW2806
AENO
MOVW   VW40, VW2808
Network 16
LD     Always_On:SM0.0
BMW    补压压力:VW2008, VW2814, 4
Network 17
LD     Always_On:SM0.0
MOVW   1组对拉位移最小值:VW2304, VW2830
AENO
MOVW   B1目标压力:VW2310, VW2832
AENO
MOVW   B2目标压力:VW2314, VW2834
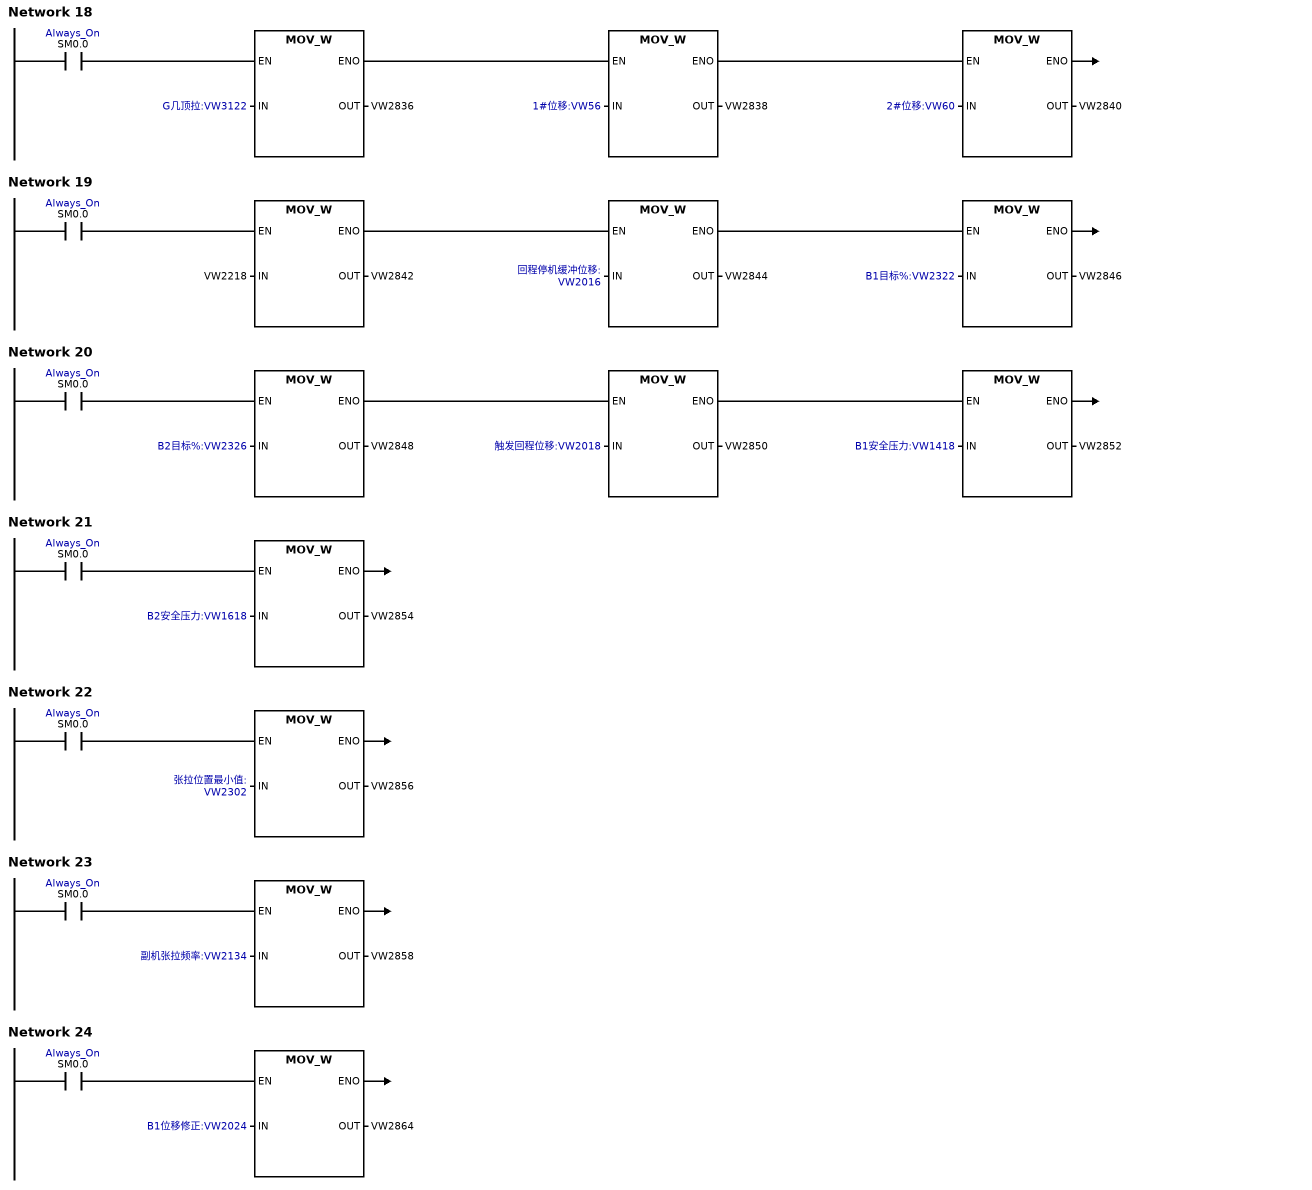
Network 18
LD     Always_On:SM0.0
MOVW   G几顶拉:VW3122, VW2836
AENO
MOVW   1#位移:VW56, VW2838
AENO
MOVW   2#位移:VW60, VW2840
Network 19
LD     Always_On:SM0.0
MOVW   VW2218, VW2842
AENO
MOVW   回程停机缓冲位移:VW2016, VW2844
AENO
MOVW   B1目标%:VW2322, VW2846
Network 20
LD     Always_On:SM0.0
MOVW   B2目标%:VW2326, VW2848
AENO
MOVW   触发回程位移:VW2018, VW2850
AENO
MOVW   B1安全压力:VW1418, VW2852
Network 21
LD     Always_On:SM0.0
MOVW   B2安全压力:VW1618, VW2854
Network 22
LD     Always_On:SM0.0
MOVW   张拉位置最小值:VW2302, VW2856
Network 23
LD     Always_On:SM0.0
MOVW   副机张拉频率:VW2134, VW2858
Network 24
LD     Always_On:SM0.0
MOVW   B1位移修正:VW2024, VW2864
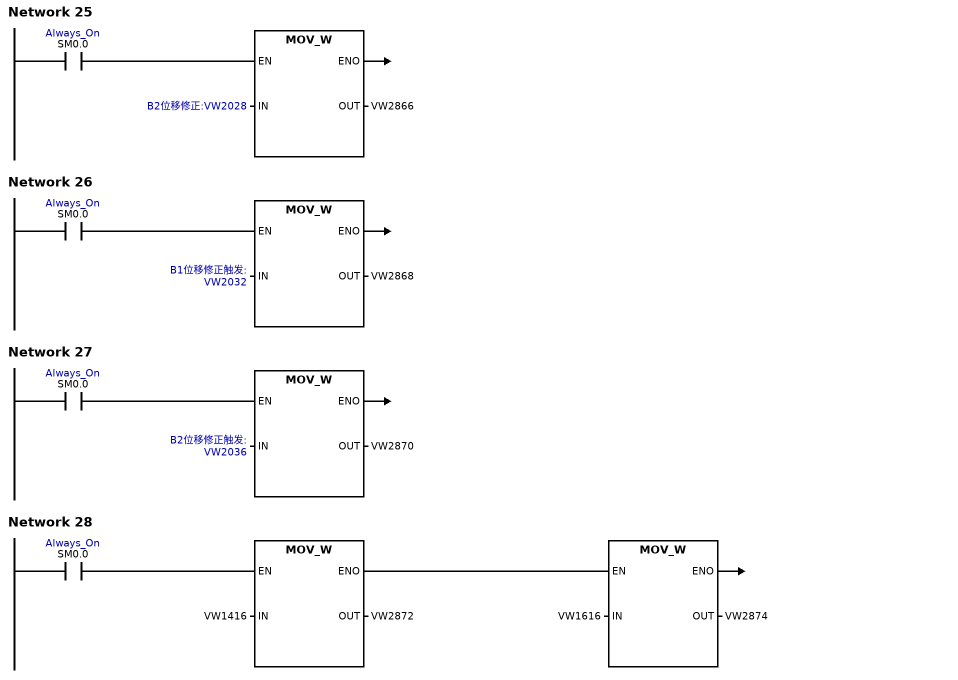
Network 25
LD     Always_On:SM0.0
MOVW   B2位移修正:VW2028, VW2866
Network 26
LD     Always_On:SM0.0
MOVW   B1位移修正触发:VW2032, VW2868
Network 27
LD     Always_On:SM0.0
MOVW   B2位移修正触发:VW2036, VW2870
Network 28
LD     Always_On:SM0.0
MOVW   VW1416, VW2872
AENO
MOVW   VW1616, VW2874
END_SUBROUTINE_BLOCK

SUBROUTINE_BLOCK 公共显示:SBR24
TITLE=子程序注释
BEGIN
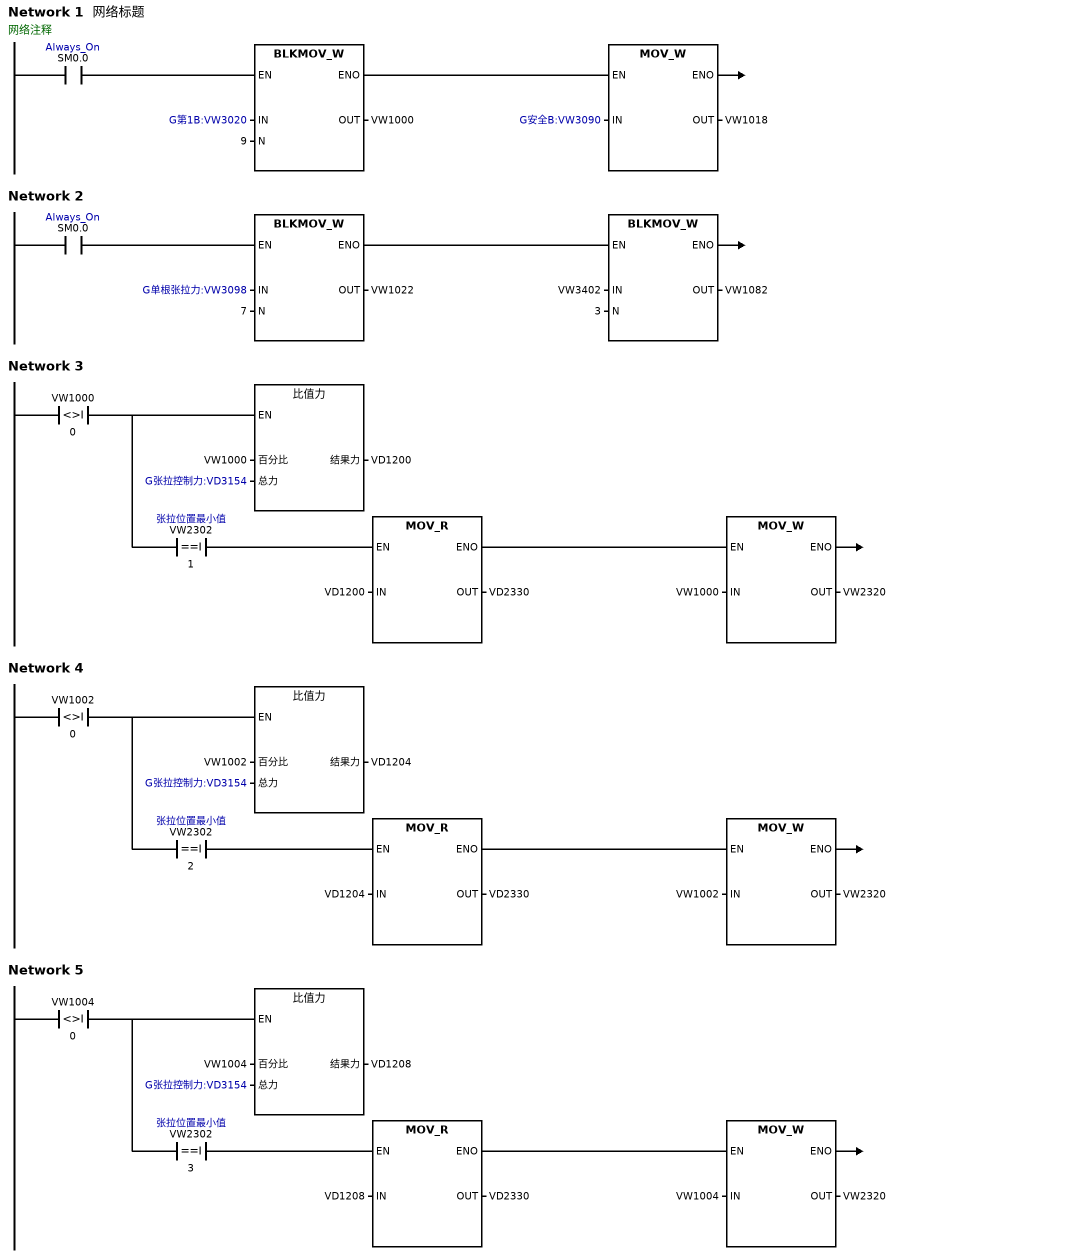
Network 1 // 网络标题
// 网络注释
LD     Always_On:SM0.0
BMW    G第1B:VW3020, VW1000, 9
AENO
MOVW   G安全B:VW3090, VW1018
Network 2
LD     Always_On:SM0.0
BMW    G单根张拉力:VW3098, VW1022, 7
AENO
BMW    VW3402, VW1082, 3
Network 3
LDW<>  VW1000, 0
CALL   比值力:SBR25, VW1000, G张拉控制力:VD3154, VD1200
AW=    张拉位置最小值:VW2302, 1
MOVR   VD1200, VD2330
AENO
MOVW   VW1000, VW2320
Network 4
LDW<>  VW1002, 0
CALL   比值力:SBR25, VW1002, G张拉控制力:VD3154, VD1204
AW=    张拉位置最小值:VW2302, 2
MOVR   VD1204, VD2330
AENO
MOVW   VW1002, VW2320
Network 5
LDW<>  VW1004, 0
CALL   比值力:SBR25, VW1004, G张拉控制力:VD3154, VD1208
AW=    张拉位置最小值:VW2302, 3
MOVR   VD1208, VD2330
AENO
MOVW   VW1004, VW2320
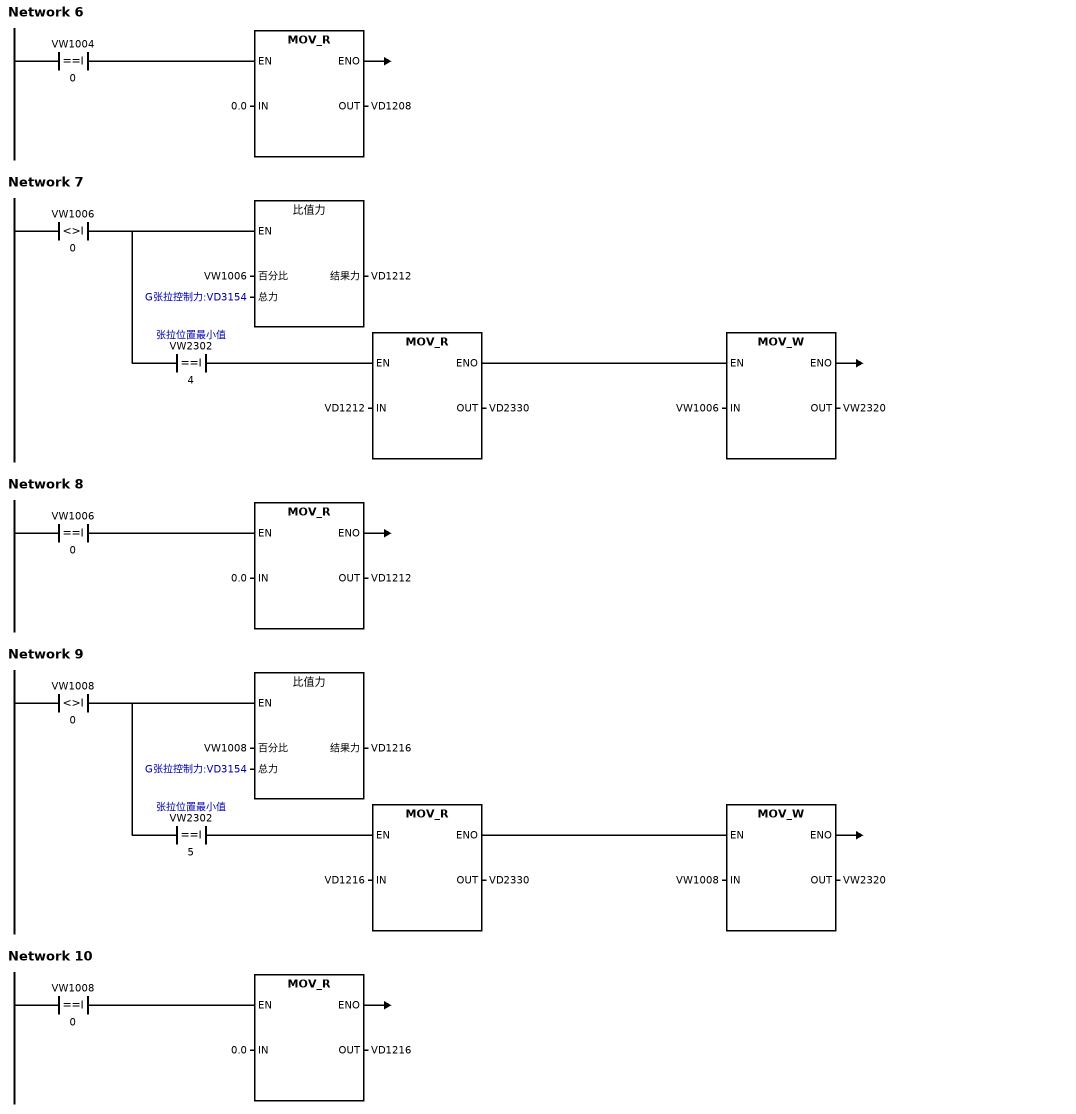
Network 6
LDW=   VW1004, 0
MOVR   0.0, VD1208
Network 7
LDW<>  VW1006, 0
CALL   比值力:SBR25, VW1006, G张拉控制力:VD3154, VD1212
AW=    张拉位置最小值:VW2302, 4
MOVR   VD1212, VD2330
AENO
MOVW   VW1006, VW2320
Network 8
LDW=   VW1006, 0
MOVR   0.0, VD1212
Network 9
LDW<>  VW1008, 0
CALL   比值力:SBR25, VW1008, G张拉控制力:VD3154, VD1216
AW=    张拉位置最小值:VW2302, 5
MOVR   VD1216, VD2330
AENO
MOVW   VW1008, VW2320
Network 10
LDW=   VW1008, 0
MOVR   0.0, VD1216
